FUNCTION isDateTimeEqual : bool
VAR_INPUT
	D1 : PtDateTime;
	D2 : PtDateTime;
END_VAR
VAR
END_VAR

isDateTimeEqual 
:= D1.Year = D2.Year
AND D1.Month = D2.Month
AND D1.Day = D2.Day
AND D1.Hour = D2.Hour
AND D1.Minute = D2.Minute
AND D1.Second = D2.Second
AND D1.Microsecond = D2.Microsecond
AND D1.TimeZone = D2.TimeZone;

END_FUNCTION

(* stored: Version 1.1.0.1, ProductVersion 3.1.4024.12
   POU isDateTimeEqual: Id {6b8bef06-2528-44df-a88b-d27ecb182c17}, SpecialFunc None *)
